TYPE ERROR :
STRUCT
	bError : BOOL;
	nErrorCode : UDINT;
	dtCurrentTime : DT;
END_STRUCT
END_TYPE

(* stored: Version 1.1.0.1
   DUT ERROR: Id {a120fa65-10d4-4ab4-a735-57ffb890ea80} *)
